TYPE CPoint :
STRUCT
	Value:LREAL;
	Base: LREAL;
END_STRUCT
END_TYPE

(* stored: Version 1.1.0.1, ProductVersion 3.1.4024.6
   DUT CPoint: Id {a1587c52-6a44-4766-a22e-1f5cf85d91d0} *)
